//Dozowniki gotowe po jakiejkolwiek zmianie i któryś jest wybrany
VIS.bDispencersSyncReady :=	NOT tofDispencersSync.Q AND 
							(fbDispencer1Sync.bOut OR fbDispencer2Sync.bOut OR fbDispencer3Sync.bOut OR fbDispencer4Sync.bOut) AND
							(eDispencer1State = E_Station.eManualMovement OR NOT fbDispencer1Sync.bOut) AND
							(eDispencer2State = E_Station.eManualMovement OR NOT fbDispencer2Sync.bOut) AND
							(eDispencer3State = E_Station.eManualMovement OR NOT fbDispencer3Sync.bOut) AND
							(eDispencer4State = E_Station.eManualMovement OR NOT fbDispencer4Sync.bOut) 	
;
//Ustawianie dozowników
IF rtDispencer1Sync.Q THEN	bDispencer1DoSync	:= TRUE;END_IF
IF rtDispencer2Sync.Q THEN	bDispencer2DoSync	:= TRUE;END_IF
IF rtDispencer3Sync.Q THEN	bDispencer3DoSync	:= TRUE;END_IF
IF rtDispencer4Sync.Q THEN	bDispencer4DoSync	:= TRUE;END_IF

//Tylko w trybie serwisowym
IF bManualMode THEN
	
	IF VIS.bDispencersSyncReady THEN
	
		//Do wszystkich
		VIS.bDispencersHoming;	
		VIS.bDispencersManualDropCatcher;
		
		//Mycie
		VIS.bDispencer12Cleaning					:=	VIS.bDispencersCleaning						AND fbDispencer1Sync.bOut AND fbDispencer2Sync.bOut;
		VIS.bDispencer34Cleaning					:=	VIS.bDispencersCleaning						AND fbDispencer3Sync.bOut AND fbDispencer4Sync.bOut;

		//Podnośnik dozownika 1
		VIS.bDispencer12ManualLifterUp       		:=	VIS.bDispencersManualLifterUp       		AND (fbDispencer1Sync.bOut OR fbDispencer2Sync.bOut);		
		VIS.bDispencer12ManualLifterDown   			:=	VIS.bDispencersManualLifterDown   			AND (fbDispencer1Sync.bOut OR fbDispencer2Sync.bOut);	
		VIS.bDispencer12LifterStepMode				:=	VIS.bDispencersLifterStepMode				;	
		IF rtHeightSetDispencer12.Q THEN
			VIS.bDispencer12LifterHeightSet         :=	TRUE;
		END_IF		                                		

		//Dozownik 1	
		VIS.bDispencer1Dose                			:=	VIS.bDispencersDose                			AND fbDispencer1Sync.bOut;		
		VIS.bDispencer1IgnoreErrors        			:=	VIS.bDispencersIgnoreErrors        			AND fbDispencer1Sync.bOut;				
		VIS.bDispencer1ManualPistonBack     		:=	VIS.bDispencersManualPistonBack     		AND fbDispencer1Sync.bOut;		
		VIS.bDispencer1ManualPistonForward  		:=	VIS.bDispencersManualPistonForward  		AND fbDispencer1Sync.bOut;
		IF fbDispencer1Sync.bOut THEN					VIS.lrDispencersActPos 							:= VIS.lrDispencer1ActPos; 			END_IF
		IF fbDispencer1Sync.bOut THEN					VIS.lrDispencersLifterActPos      				:=	VIS.lrDispencer12LifterActPos ; END_IF	
		VIS.bDispencer1PullingFast          		:=	VIS.bDispencersPullingFast          		AND fbDispencer1Sync.bOut;		
		VIS.bDispencer1PullingSlow         			:=	VIS.bDispencersPullingSlow         			AND fbDispencer1Sync.bOut;		
		VIS.bDispencer1ManualSuckValve     			:=	VIS.bDispencersManualSuckValve     			AND fbDispencer1Sync.bOut;		
		VIS.bDispencer1ManualDoseValve     			:=	VIS.bDispencersManualDoseValve     			AND fbDispencer1Sync.bOut;
		VIS.lrDispencer12LifterSetPosStepMode		:=	VIS.lrDispencersLifterSetPosStepMode;	
		//Ready position					    	:=	//Ready position					    	AND fbDispencer1Sync.bOut;		

		//Dozownik 2 	
		VIS.bDispencer2Dose                			:=	VIS.bDispencersDose                			AND fbDispencer2Sync.bOut;		
		VIS.bDispencer2IgnoreErrors        			:=	VIS.bDispencersIgnoreErrors        			AND fbDispencer2Sync.bOut;				
		VIS.bDispencer2ManualPistonBack     		:=	VIS.bDispencersManualPistonBack     		AND fbDispencer2Sync.bOut;		
		VIS.bDispencer2ManualPistonForward  		:=	VIS.bDispencersManualPistonForward  		AND fbDispencer2Sync.bOut;
		IF fbDispencer2Sync.bOut THEN					VIS.lrDispencersActPos 							:= VIS.lrDispencer2ActPos; 			END_IF
		IF fbDispencer2Sync.bOut THEN					VIS.lrDispencersLifterActPos      				:=	VIS.lrDispencer12LifterActPos ; END_IF	
		VIS.bDispencer2PullingFast          		:=	VIS.bDispencersPullingFast          		AND fbDispencer2Sync.bOut;		
		VIS.bDispencer2PullingSlow         			:=	VIS.bDispencersPullingSlow         			AND fbDispencer2Sync.bOut;		
		VIS.bDispencer2ManualSuckValve     			:=	VIS.bDispencersManualSuckValve     			AND fbDispencer2Sync.bOut;		
		VIS.bDispencer2ManualDoseValve     			:=	VIS.bDispencersManualDoseValve     			AND fbDispencer2Sync.bOut;
		VIS.lrDispencer12LifterSetPosStepMode		:=	VIS.lrDispencersLifterSetPosStepMode;	                 
		//Ready position					    	:=	//Ready position					    	AND fbDispencer2Sync.bOut;		
		
		//Podnośnik dozownika 34
		VIS.bDispencer34ManualLifterUp       		:=	VIS.bDispencersManualLifterUp       		AND (fbDispencer3Sync.bOut OR fbDispencer4Sync.bOut);		
		VIS.bDispencer34ManualLifterDown   			:=	VIS.bDispencersManualLifterDown   			AND (fbDispencer3Sync.bOut OR fbDispencer4Sync.bOut);	
		VIS.bDispencer34LifterStepMode				:=	VIS.bDispencersLifterStepMode				;		
		IF rtHeightSetDispencer34.Q THEN
			VIS.bDispencer34LifterHeightSet         :=	TRUE;
		END_IF		
		//Dozownik 3 	
		VIS.bDispencer3Dose                			:=	VIS.bDispencersDose                			AND fbDispencer3Sync.bOut;		
		VIS.bDispencer3IgnoreErrors        			:=	VIS.bDispencersIgnoreErrors        			AND fbDispencer3Sync.bOut;				
		VIS.bDispencer3ManualPistonBack     		:=	VIS.bDispencersManualPistonBack     		AND fbDispencer3Sync.bOut;		
		VIS.bDispencer3ManualPistonForward  		:=	VIS.bDispencersManualPistonForward  		AND fbDispencer3Sync.bOut;
		IF fbDispencer3Sync.bOut THEN					VIS.lrDispencersActPos 							:= VIS.lrDispencer3ActPos; 			END_IF
		IF fbDispencer3Sync.bOut THEN					VIS.lrDispencersLifterActPos      				:=	VIS.lrDispencer34LifterActPos ; END_IF	
		VIS.bDispencer3PullingFast          		:=	VIS.bDispencersPullingFast          		AND fbDispencer3Sync.bOut;		
		VIS.bDispencer3PullingSlow         			:=	VIS.bDispencersPullingSlow         			AND fbDispencer3Sync.bOut;		
		VIS.bDispencer3ManualSuckValve     			:=	VIS.bDispencersManualSuckValve     			AND fbDispencer3Sync.bOut;		
		VIS.bDispencer3ManualDoseValve     			:=	VIS.bDispencersManualDoseValve     			AND fbDispencer3Sync.bOut;
		VIS.lrDispencer34LifterSetPosStepMode		:=	VIS.lrDispencersLifterSetPosStepMode;	                 
		//Ready position					    	:=	//Ready position					    	AND fbDispencer3Sync.bOut;		
	                           		
		//Dozownik 4 	
		VIS.bDispencer4Dose                			:=	VIS.bDispencersDose                			AND fbDispencer4Sync.bOut;		
		VIS.bDispencer4IgnoreErrors        			:=	VIS.bDispencersIgnoreErrors        			AND fbDispencer4Sync.bOut;				
		VIS.bDispencer4ManualPistonBack     		:=	VIS.bDispencersManualPistonBack     		AND fbDispencer4Sync.bOut;		
		VIS.bDispencer4ManualPistonForward  		:=	VIS.bDispencersManualPistonForward  		AND fbDispencer4Sync.bOut;
		IF fbDispencer4Sync.bOut THEN					VIS.lrDispencersActPos 							:= VIS.lrDispencer4ActPos; 			END_IF
		IF fbDispencer4Sync.bOut THEN					VIS.lrDispencersLifterActPos      				:=	VIS.lrDispencer34LifterActPos ; END_IF	
		VIS.bDispencer4PullingFast          		:=	VIS.bDispencersPullingFast          		AND fbDispencer4Sync.bOut;		
		VIS.bDispencer4PullingSlow         			:=	VIS.bDispencersPullingSlow         			AND fbDispencer4Sync.bOut;		
		VIS.bDispencer4ManualSuckValve     			:=	VIS.bDispencersManualSuckValve     			AND fbDispencer4Sync.bOut;		
		VIS.bDispencer4ManualDoseValve     			:=	VIS.bDispencersManualDoseValve     			AND fbDispencer4Sync.bOut;
		VIS.lrDispencer34LifterSetPosStepMode		:=	VIS.lrDispencersLifterSetPosStepMode;	                 
		//Ready position					    	:=	//Ready position					    	AND fbDispencer4Sync.bOut;		
			
	ELSE
		
		VIS.bDispencer1Dose                			:=	VIS.bDispencersDose    					 := FALSE;            			
		VIS.bDispencer1ManualPistonBack     		:=	VIS.bDispencersManualPistonBack     	 := FALSE;  
		VIS.bDispencer1ManualPistonForward  		:=	VIS.bDispencersManualPistonForward  	 := FALSE;  
		VIS.lrDispencersActPos 						:=	1234;			
		VIS.bDispencer12ManualLifterUp       		:=	VIS.bDispencersManualLifterUp       	 := FALSE;  	
		VIS.bDispencer12ManualLifterDown   			:=	VIS.bDispencersManualLifterDown   		 := FALSE;  
		VIS.lrDispencersLifterActPos      			:=	1234;		
		VIS.bDispencer1PullingFast          		:=	VIS.bDispencersPullingFast          	 := FALSE;  
		VIS.bDispencer1PullingSlow         			:=	VIS.bDispencersPullingSlow         		 := FALSE;  
		VIS.bDispencer1ManualSuckValve     			:=	VIS.bDispencersManualSuckValve     		 := FALSE;  
		VIS.bDispencer1ManualDoseValve     			:=	VIS.bDispencersManualDoseValve     		 := FALSE;  
		VIS.lrDispencer12LifterSetPosStepMode		:=	VIS.lrDispencersLifterSetPosStepMode	 := 2;	
		VIS.bDispencer12LifterStepMode				:=	VIS.bDispencersLifterStepMode		 	 := FALSE;  	
		//Ready position					    	:=	//Ready position					    
		//nie nadpisywać (bazownaie) VIS.bDispencer12LifterHeightSet          			:=	VIS.bDispencersHeightSet          		 := FALSE;  
		
		VIS.bDispencer2Dose                			:=	VIS.bDispencersDose    					 := FALSE;            			
		VIS.bDispencer2ManualPistonBack     		:=	VIS.bDispencersManualPistonBack     	 := FALSE;  
		VIS.bDispencer2ManualPistonForward  		:=	VIS.bDispencersManualPistonForward  	 := FALSE;  
		VIS.lrDispencersActPos 						:=	1234;			
		VIS.bDispencer12ManualLifterUp       		:=	VIS.bDispencersManualLifterUp       	 := FALSE;  	
		VIS.bDispencer12ManualLifterDown   			:=	VIS.bDispencersManualLifterDown   		 := FALSE;  
		VIS.lrDispencersLifterActPos      			:=	1234;		
		VIS.bDispencer2PullingFast          		:=	VIS.bDispencersPullingFast          	 := FALSE;  
		VIS.bDispencer2PullingSlow         			:=	VIS.bDispencersPullingSlow         		 := FALSE;  
		VIS.bDispencer2ManualSuckValve     			:=	VIS.bDispencersManualSuckValve     		 := FALSE;  
		VIS.bDispencer2ManualDoseValve     			:=	VIS.bDispencersManualDoseValve     		 := FALSE;  
		VIS.lrDispencer12LifterSetPosStepMode		:=	VIS.lrDispencersLifterSetPosStepMode	 := 2;	
		VIS.bDispencer12LifterStepMode				:=	VIS.bDispencersLifterStepMode		 	 := FALSE;  	
		//Ready position					    	:=	//Ready position					    
		 		
		VIS.bDispencer3Dose                			:=	VIS.bDispencersDose   					 := FALSE;            			
		VIS.bDispencer3ManualPistonBack     		:=	VIS.bDispencersManualPistonBack     	 := FALSE;  
		VIS.bDispencer3ManualPistonForward  		:=	VIS.bDispencersManualPistonForward  	 := FALSE;  
		VIS.lrDispencersActPos 						:=	1234;			
		VIS.bDispencer34ManualLifterUp       		:=	VIS.bDispencersManualLifterUp       	 := FALSE;  	
		VIS.bDispencer34ManualLifterDown   			:=	VIS.bDispencersManualLifterDown   		 := FALSE;  
		VIS.lrDispencersLifterActPos      			:=	1234;		
		VIS.bDispencer3PullingFast          		:=	VIS.bDispencersPullingFast          	 := FALSE;  
		VIS.bDispencer3PullingSlow         			:=	VIS.bDispencersPullingSlow         		 := FALSE;  
		VIS.bDispencer3ManualSuckValve     			:=	VIS.bDispencersManualSuckValve     		 := FALSE;  
		VIS.bDispencer3ManualDoseValve     			:=	VIS.bDispencersManualDoseValve     		 := FALSE;  
		VIS.lrDispencer34LifterSetPosStepMode		:=	VIS.lrDispencersLifterSetPosStepMode	 := 2;	
		VIS.bDispencer34LifterStepMode				:=	VIS.bDispencersLifterStepMode		 	 := FALSE;  	
		//Ready position					    	:=	//Ready position					    
		//VIS.bDispencer34LifterHeightSet          	:=	VIS.bDispencersHeightSet          		 := FALSE;  

		VIS.bDispencer4Dose                			:=	VIS.bDispencersDose    					 := FALSE;            			
		VIS.bDispencer4ManualPistonBack     		:=	VIS.bDispencersManualPistonBack     	 := FALSE;  
		VIS.bDispencer4ManualPistonForward  		:=	VIS.bDispencersManualPistonForward  	 := FALSE;  
		VIS.lrDispencersActPos 						:=	1234;			
		VIS.bDispencer34ManualLifterUp       		:=	VIS.bDispencersManualLifterUp       	 := FALSE;  	
		VIS.bDispencer34ManualLifterDown   			:=	VIS.bDispencersManualLifterDown   		 := FALSE;  
		VIS.lrDispencersLifterActPos      			:=	1234;		
		VIS.bDispencer4PullingFast          		:=	VIS.bDispencersPullingFast          	 := FALSE;  
		VIS.bDispencer4PullingSlow         			:=	VIS.bDispencersPullingSlow         		 := FALSE;  
		VIS.bDispencer4ManualSuckValve     			:=	VIS.bDispencersManualSuckValve     		 := FALSE;  
		VIS.bDispencer4ManualDoseValve     			:=	VIS.bDispencersManualDoseValve     		 := FALSE;  
		VIS.lrDispencer34LifterSetPosStepMode		:=	VIS.lrDispencersLifterSetPosStepMode	 := 2;	
		VIS.bDispencer34LifterStepMode				:=	VIS.bDispencersLifterStepMode		 	 := FALSE;  	
		//Ready position					    	:=	//Ready position					    
		
	END_IF
	
END_IF


(********KASOWANIE ROZKAZÓW CYKLI*********)
IF fbDispencer1.bCycleDone AND bManualMode AND
	(NOT fbDispencer2Sync.bOut AND NOT fbDispencer3Sync.bOut AND NOT fbDispencer4Sync.bOut)
THEN
    VIS.bDispencer1Dose := VIS.bDispencersDose :=  FALSE;
END_IF

IF fbDispencer2.bCycleDone AND bManualMode AND
	(NOT fbDispencer1Sync.bOut AND NOT fbDispencer3Sync.bOut AND NOT fbDispencer4Sync.bOut)
THEN
    VIS.bDispencer2Dose		:= VIS.bDispencersDose := FALSE;
END_IF

IF fbDispencer3.bCycleDone AND bManualMode AND
	(NOT fbDispencer1Sync.bOut AND NOT fbDispencer2Sync.bOut AND NOT fbDispencer4Sync.bOut)
THEN
    VIS.bDispencer3Dose		:= VIS.bDispencersDose := FALSE;
END_IF

IF fbDispencer4.bCycleDone AND bManualMode AND
	(NOT fbDispencer1Sync.bOut AND NOT fbDispencer2Sync.bOut AND NOT fbDispencer3Sync.bOut)

THEN
    VIS.bDispencer4Dose	:= VIS.bDispencersDose := FALSE;
END_IF
IF fbDispencer1.bCycleDone AND  fbDispencer2.bCycleDone AND NOT fbDispencer3.bCycleDone AND NOT fbDispencer4.bCycleDone AND bManualMode AND
	(fbDispencer1Sync.bOut AND fbDispencer2Sync.bOut AND NOT fbDispencer3Sync.bOut AND NOT fbDispencer4Sync.bOut)
THEN
    VIS.bDispencersDose :=  FALSE;
END_IF
IF NOT fbDispencer1.bCycleDone AND  NOT fbDispencer2.bCycleDone AND fbDispencer3.bCycleDone AND fbDispencer4.bCycleDone AND bManualMode AND
	(NOT fbDispencer1Sync.bOut AND NOT fbDispencer2Sync.bOut AND fbDispencer3Sync.bOut AND fbDispencer4Sync.bOut)
THEN
    VIS.bDispencersDose :=  FALSE;
END_IF
IF fbDispencer1.bCycleDone AND  fbDispencer2.bCycleDone AND  fbDispencer3.bCycleDone AND  fbDispencer4.bCycleDone AND bManualMode AND
	(fbDispencer1Sync.bOut AND fbDispencer2Sync.bOut AND fbDispencer3Sync.bOut AND fbDispencer4Sync.bOut)
THEN
    VIS.bDispencersDose :=  FALSE;
END_IF


(*****KONIEC KASOWANIA ROZKAZÓW CYKLI*****)
END_ACTION

ACTION aDosingChartHMI:
 fbDosingChart1(
	bWrite:= VIS.bDispencer1Dose, 
	nCycleTime:= 5, 
	lrData1:= VIS.lrDispencer1ActPos, 
	lrData2:= VIS.lrDispencer12LifterActPos, 
	bData3:= P02_Dispencers.QbDispencer1SuckingValveActuator, 
	bData4:= P02_Dispencers.QbDispencer1DosingValveActuator,
	bData5:= P02_Dispencers.QbDispencer1DropCatcherValveActuator,
	AsData=>VIS.AsChartDose1 );
	
 fbDosingStChart1(
	bWrite:= VIS.bDispencer1Dose, 
	udiCycleTime:= 5,
	lrAiData0:= VIS.lrDispencer1ActPos,
	lrAiData1:= VIS.lrDispencer12LifterActPos, 
	lrAiData2:= BOOL_TO_LREAL(P02_Dispencers.QbDispencer1SuckingValveActuator),
	lrAiData3:= BOOL_TO_LREAL(P02_Dispencers.QbDispencer1DosingValveActuator), 
	lrAiData4:= BOOL_TO_LREAL(P02_Dispencers.QbDispencer1DropCatcherValveActuator), 
	AiData=> VIS.AStAsChartDose1[0] );

fbDosingChart2(
	bWrite:= VIS.bDispencer2Dose, 
	nCycleTime:= 5, 
	lrData1:= VIS.lrDispencer2ActPos, 
	lrData2:= VIS.lrDispencer12LifterActPos, 
	bData3:= P02_Dispencers.QbDispencer2SuckingValveActuator, 
	bData4:= P02_Dispencers.QbDispencer2DosingValveActuator,
	bData5:= P02_Dispencers.QbDispencer2DropCatcherValveActuator,
	AsData=>VIS.AsChartDose2 );

 fbDosingStChart2(
	bWrite:= VIS.bDispencer1Dose, 
	udiCycleTime:= 5,
	lrAiData0:= VIS.lrDispencer2ActPos,
	lrAiData1:= VIS.lrDispencer12LifterActPos, 
	lrAiData2:= BOOL_TO_LREAL(P02_Dispencers.QbDispencer2SuckingValveActuator),
	lrAiData3:= BOOL_TO_LREAL(P02_Dispencers.QbDispencer2DosingValveActuator), 
	lrAiData4:= BOOL_TO_LREAL(P02_Dispencers.QbDispencer2DropCatcherValveActuator), 
	AiData=> VIS.AStAsChartDose2[0] );
	
fbDosingChart3(
	bWrite:= VIS.bDispencer3Dose, 
	nCycleTime:= 5,//nChartCycleTime, 
	lrData1:= VIS.lrDispencer3ActPos, 
	lrData2:= VIS.lrDispencer34LifterActPos, 
	bData3:= P02_Dispencers.QbDispencer3SuckingValveActuator, 
	bData4:= P02_Dispencers.QbDispencer3DosingValveActuator,
	bData5:= P02_Dispencers.QbDispencer3DropCatcherValveActuator,
	AsData=>VIS.AsChartDose3 );
	
 fbDosingStChart3(
	bWrite:= VIS.bDispencer1Dose, 
	udiCycleTime:= 5,
	lrAiData0:= VIS.lrDispencer3ActPos,
	lrAiData1:= VIS.lrDispencer34LifterActPos, 
	lrAiData2:= BOOL_TO_LREAL(P02_Dispencers.QbDispencer3SuckingValveActuator),
	lrAiData3:= BOOL_TO_LREAL(P02_Dispencers.QbDispencer3DosingValveActuator), 
	lrAiData4:= BOOL_TO_LREAL(P02_Dispencers.QbDispencer3DropCatcherValveActuator), 
	AiData=> VIS.AStAsChartDose3[0] );

fbDosingChart4(
	bWrite:= VIS.bDispencer4Dose, 
	nCycleTime:= 5,//nChartCycleTime, 
	lrData1:= VIS.lrDispencer4ActPos, 
	lrData2:= VIS.lrDispencer34LifterActPos, 
	bData3:= P02_Dispencers.QbDispencer4SuckingValveActuator, 
	bData4:= P02_Dispencers.QbDispencer4DosingValveActuator,
	bData5:= P02_Dispencers.QbDispencer4DropCatcherValveActuator,
	AsData=>VIS.AsChartDose4 );

fbDosingStChart4(
	bWrite:= VIS.bDispencer1Dose, 
	udiCycleTime:= 5,
	lrAiData0:= VIS.lrDispencer4ActPos,
	lrAiData1:= VIS.lrDispencer34LifterActPos, 
	lrAiData2:= BOOL_TO_LREAL(P02_Dispencers.QbDispencer4SuckingValveActuator),
	lrAiData3:= BOOL_TO_LREAL(P02_Dispencers.QbDispencer4DosingValveActuator), 
	lrAiData4:= BOOL_TO_LREAL(P02_Dispencers.QbDispencer4DropCatcherValveActuator), 
	AiData=> VIS.AStAsChartDose4[0] );
END_ACTION

ACTION aDropCatcher:
(**Uruchamianie ssawki tacek**)
P02_Dispencers.QbDispencerDropCatcherSuck;
IF (P00_PackML.fbPMLAuto.ePMLState = E_PMLState.ePMLState_EXECUTE OR P00_PackML.fbPMLModeManager.eModeStatus = E_PMLUnitMode.ePMLUnitMode_MANUAL) THEN
	fbDropCatcherSuck(T1:=T#5S , T0:=T#30S , Q=>P02_Dispencers.QbDispencerDropCatcherSuck);
	;
ELSE
	P02_Dispencers.QbDispencerDropCatcherSuck := FALSE;
END_IF

IF VIS.bDispencerManualDropCatcherSuck AND bManualMode THEN
	
	P02_Dispencers.QbDispencerDropCatcherSuck	:= TRUE;
END_IF
END_ACTION

ACTION aExSensor:


(** Czujnik Ex w zbiorniku **)

tonLowLevelExSensor(IN:=NOT IbTankLevelHighEX AND IbTankLevelLowEX AND NOT tonErrorExSensorDelay.Q AND bExEnable, PT:=T#1S);

IF tonLowLevelExSensor.Q THEN
	bTank1LevelExSensor:=TRUE;
ELSE
	bTank1LevelExSensor:=FALSE;
END_IF





//Błąd czujnika Ex
tonErrorExSensorDelay(IN:=IbTankLevelExError, PT:=T#5S);

IF tonErrorExSensorDelay.Q AND NOT TanksError.bError AND bExEnable AND bTank1SupplyPumpEnable THEN
	TanksError.bError:=TRUE;
	TanksError.bReset:=FALSE;
	TanksError.udiStationID:=78;
	TanksError.nErrorCode:=368;
	TanksError.sStationName:='Błąd systemu';
	TanksError.sErrorString:='Błąd czujnika poziomu Ex w zbiorniku. Sprawdz podłączenie lub stan separatora';
END_IF
END_ACTION

ACTION aLevelSensorCalibration:


(*
	bDialogBoxOn:BOOL;						(**)		// Wyświetlanie okienka komunikatów
	bDialogBoxText:STRING;					(**)		// Treść na oknie komunikatów
	bDialogBoxAck:BOOL;						(*t*)		// Potwierdzenie ogólne
	bDialogBoxCancelAck:BOOL;				(*t*)		// Wycofywanie procedury
	nDialogBoxType:UINT;								// Rodzaj okna, 0-nic, 1-tylko przysisk OK, 2 - tylko przycisk Anuluj, 3 - Przycisk OK i Anuluj
*)


(****Kalibracja czujnika nr 1 na pusto****)
tonTankLevelSensorCalibrationLight(IN:= nCalibrationDialog = 1 AND (VIS.bTank1LevelSensorCalibrationLight),PT:=T#10S);
tonTankLevelSensorCalibrationDark(IN:= nCalibrationDialog = 1 AND (VIS.bTank1LevelSensorCalibrationDark), PT:=T#5S);
IF VIS.bTank1LevelSensorCalibrationLight OR VIS.bTank1LevelSensorCalibrationDark THEN 		//Rozpoczaecie procedury kalibracji
	CASE nCalibrationDialog OF
		
		0: //Pytanie Czy na pewno
			VIS.nDialogBoxType	:=	3;									//Wyświetlanie przycisku OK i Anuluj
			IF VIS.bTank1LevelSensorCalibrationLight THEN
				VIS.bDialogBoxText	:=	'Want calibrate the level sensor to an empty tank? Immerse the sensor in the mass and remove it, simulating an empty tank.';
				VIS.sDialogBoxPicture	:= 'info';
			ELSIF VIS.bTank1LevelSensorCalibrationDark THEN
				VIS.bDialogBoxText	:=	'Should I calibrate the level sensor to a full tank? Immerse the sensor in the mass to simulate a full tank.';
				VIS.sDialogBoxPicture	:= 'info';
			END_IF
			VIS.bDialogBoxOn	:=	TRUE;
			IF VIS.bDialogBoxAck THEN
				VIS.bDialogBoxAck	:=	FALSE;		
				nCalibrationDialog:=nCalibrationDialog+1;
			ELSIF VIS.bDialogBoxCancelAck THEN
				VIS.bTank1LevelSensorCalibrationLight	:=	FALSE;
				VIS.bTank1LevelSensorCalibrationDark	:=	FALSE;

				//MAIN.aResetDialog();	
				nCalibrationDialog := 0;
			END_IF
			
		1: //Trwa kalibracja
			VIS.nDialogBoxType	:=	0;									//Bez przycisków
			
			IF VIS.bTank1LevelSensorCalibrationLight THEN
				QbTank1LevelSensorCalibration := NOT tonTankLevelSensorCalibrationLight.Q;	
				VIS.bDialogBoxText	:=	'Empty tank calibration in progress 1...';
				VIS.sDialogBoxPicture	:= '';
			END_IF
			IF VIS.bTank1LevelSensorCalibrationDark THEN
				QbTank1LevelSensorCalibration := NOT tonTankLevelSensorCalibrationDark.Q;	
				VIS.bDialogBoxText	:=	'Full tank calibration in progress 1...';
				VIS.sDialogBoxPicture	:= '';
			END_IF
			IF tonTankLevelSensorCalibrationLight.Q OR tonTankLevelSensorCalibrationDark.Q THEN
				nCalibrationDialog:=nCalibrationDialog+1;
			END_IF
			
		2: //Koniec kalibracji
			VIS.nDialogBoxType	:=	1;									//Potwierdz kalibracje
			VIS.bDialogBoxText	:=	'Calibration completed successfully';
			VIS.sDialogBoxPicture	:= 'ok';
			IF VIS.bTank1LevelSensorCalibrationLight OR VIS.bTank1LevelSensorCalibrationDark THEN
				bTank1LevelSensorCalibrated := TRUE;						//Zmienna presistent o kalibracji
			END_IF
			
			IF  VIS.bDialogBoxAck THEN
				VIS.bDialogBoxAck :=					FALSE;
				VIS.bTank1LevelSensorCalibrationLight	:=	FALSE;
				VIS.bTank1LevelSensorCalibrationDark	:=	FALSE;
				P00_Visualization.aResetDialog();
				nCalibrationDialog := 0;
			END_IF
			
	END_CASE
END_IF
END_ACTION

ACTION aLimits:

(*Zabezpieczenie nastaw dozowników*)
//Dozownika 1 i 2 (1 faza)
IF VIS.lrDispencer1DoseValveOpenTimeAccShow>0 			THEN 	VIS.lrDispencer1DoseValveOpenVolumeShow		:=0;		END_IF
IF VIS.lrDispencer1DoseValveCloseTimeDecShow>0 			THEN	VIS.lrDispencer1DoseValveCloseVolumeShow	:=0;		END_IF
IF VIS.bDispencer1DoseSuckingShow 						THEN	VIS.lrDispencer1DoseValveCloseVolumeShow	:=0;		END_IF
IF VIS.lrDispencer1SuckValveOpenTimeDelayShow>0 		THEN	VIS.lrDispencer1SuckValveOpenVolumeShow		:=0;		END_IF
IF VIS.lrDispencer1SuckValveCloseTimeDelayShow>0 		THEN	VIS.lrDispencer1SuckValveCloseVolumeShow	:=0;		END_IF
IF VIS.lrDispencer1Phase1VolumeShow > VIS.lrDispencer1DoseVolumeShow - VIS.lrDispencer1Phase2VolumeShow THEN	VIS.lrDispencer1Phase1VolumeShow	:= VIS.lrDispencer1DoseVolumeShow - VIS.lrDispencer1Phase2VolumeShow;END_IF
IF VIS.lrDispencer1Phase2VolumeShow > VIS.lrDispencer1DoseVolumeShow - VIS.lrDispencer1Phase1VolumeShow THEN	VIS.lrDispencer1Phase2VolumeShow 	:= VIS.lrDispencer1DoseVolumeShow - VIS.lrDispencer1Phase1VolumeShow;END_IF
IF VIS.lrDispencer1Phase2VolumeShow > VIS.lrDispencer1DoseVolumeShow 									THEN	VIS.lrDispencer1Phase1VolumeShow	:= 0;	VIS.lrDispencer1Phase2VolumeShow 	:= VIS.lrDispencer1DoseVolumeShow;END_IF

// Dozownika 3 i 4 (2 faza)
IF VIS.lrDispencer2DoseValveOpenTimeAccShow>0 			THEN	VIS.lrDispencer2DoseValveOpenVolumeShow		:=0;		END_IF
IF VIS.lrDispencer2DoseValveCloseTimeDecShow>0 			THEN	VIS.lrDispencer2DoseValveCloseVolumeShow	:=0;		END_IF
IF VIS.bDispencer2DoseSuckingShow 						THEN	VIS.lrDispencer2DoseValveCloseVolumeShow	:=0;		END_IF
IF VIS.lrDispencer2SuckValveOpenTimeDelayShow>0 		THEN	VIS.lrDispencer2SuckValveOpenVolumeShow		:=0;		END_IF
IF VIS.lrDispencer2SuckValveCloseTimeDelayShow>0 		THEN	VIS.lrDispencer2SuckValveCloseVolumeShow	:=0;		END_IF
IF VIS.lrDispencer2Phase1VolumeShow > VIS.lrDispencer2DoseVolumeShow - VIS.lrDispencer2Phase2VolumeShow THEN	VIS.lrDispencer2Phase1VolumeShow	:= VIS.lrDispencer2DoseVolumeShow - VIS.lrDispencer2Phase2VolumeShow;END_IF
IF VIS.lrDispencer2Phase2VolumeShow > VIS.lrDispencer2DoseVolumeShow - VIS.lrDispencer2Phase1VolumeShow THEN	VIS.lrDispencer2Phase2VolumeShow 	:= VIS.lrDispencer2DoseVolumeShow - VIS.lrDispencer2Phase1VolumeShow;END_IF
IF VIS.lrDispencer2Phase2VolumeShow > VIS.lrDispencer2DoseVolumeShow 									THEN	VIS.lrDispencer2Phase1VolumeShow	:= 0;	VIS.lrDispencer2Phase2VolumeShow 	:= VIS.lrDispencer2DoseVolumeShow;END_IF

IF lrDispencersLifterReadyPosition <1 					THEN	lrDispencersLifterReadyPosition			:=	270;													END_IF
IF 	VIS.lrDispencersLifterReadyPositionShow > 
	(P02_Dispencers.fbDispencer1.lrMaxPosition - 2)		THEN	VIS.lrDispencersLifterReadyPositionShow	:=	P02_Dispencers.fbDispencer1.lrMaxPosition - 2;			END_IF
	
	
IF 	VIS.lrFormsDragingLeftStartPosition		= 0		THEN	VIS.lrFormsDragingLeftStartPosition		:=	7;		END_IF;
IF 	VIS.lrFormsDragingLeftEndPosition		= 0		THEN	VIS.lrFormsDragingLeftEndPosition		:=	137;	END_IF;
IF 	VIS.lrFormsDragingRightStartPosition	= 0		THEN	VIS.lrFormsDragingRightStartPosition	:=	7.5;		END_IF;
IF 	VIS.lrFormsDragingRightEndPosition		= 0		THEN	VIS.lrFormsDragingRightEndPosition		:=	139;	END_IF;;
END_ACTION

ACTION aTankHeating:
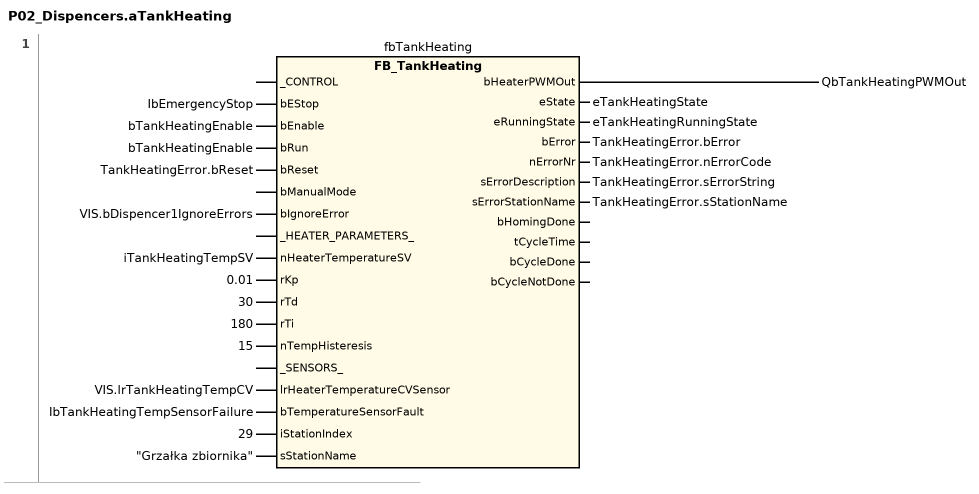
// NETWORK 1
fbTankHeating(
    bEStop := IbEmergencyStop,
    bEnable := bTankHeatingEnable,
    bRun := bTankHeatingEnable,
    bReset := TankHeatingError.bReset,
    bIgnoreError := VIS.bDispencer1IgnoreErrors,
    nHeaterTemperatureSV := iTankHeatingTempSV,
    rKp := 0.01,
    rTd := 30,
    rTi := 180,
    nTempHisteresis := 15,
    lrHeaterTemperatureCVSensor := VIS.lrTankHeatingTempCV,
    bTemperatureSensorFault := IbTankHeatingTempSensorFailure,
    iStationIndex := 29,
    sStationName := "Grzałka zbiornika",
    eState => eTankHeatingState,
    eRunningState => eTankHeatingRunningState,
    bError => TankHeatingError.bError,
    nErrorNr => TankHeatingError.nErrorCode,
    sErrorDescription => TankHeatingError.sErrorString,
    sErrorStationName => TankHeatingError.sStationName); // FB_TankHeating
QbTankHeatingPWMOut := fbTankHeating.bHeaterPWMOut;
END_ACTION

ACTION aTanks:
//Sterowanie Mieszadłem zbiornikowym
IF IbEmergencyStop (*AND IbFuseTankMixerEngineOK*) THEN
	QbTank1MixerStart:=(bTank1MixerEnable AND NOT bChangeover) OR (VIS.bTank1ManualMixer AND bManualMode);
ELSE
	QbTank1MixerStart:=FALSE;
	VIS.bTank1ManualMixer:=FALSE;
END_IF

//Sterowanie grzaniem zbiornika
//QbTank1HeaterOn:=IbEmergencyStopButton AND bTank1HeaterEnable OR (VIS.bManualTank1Heater AND bManualMode);

//Odwracanie sygnałów z czujników poziomu z receptur
bTank1LevelSignalInvert;									// Odwróć sygnał z czujnika zbiornika pierwszego
bTank2LevelSignalInvert;									// Odwróć sygnał z czujnika zbionirka drugiego
VIS.bTank1SupplyPumpEnableShow;
VIS.bTank2SupplyPumpEnableShow;
//Zmienne do poglądu zadziałania pomp od czujników
VIS.bHMITank1LevelSensorPumpOn;								// Sygnał z czujnika poziomu 1 załączający pompe 1 zależnie od ustawień (do podglądu sprawdzenia działania pompy bez jej załaczania)
VIS.bHMITank2LevelSensorPumpOn;								// Sygnał z czujnika poziomu 2 załączający pompe 2 zaleznie od ustawień (do podglądu sprawdzenia działania pompy bez jej załaczania)

//Odwracanie sygnałów z czujników poziomu
IF NOT bTank1LevelSignalInvert THEN
	bTank1LevelLow					:=	IbTank1LevelLow OR bTank1LevelLowConductiveSensor OR bTank1LevelExSensor; 	
	VIS.bHMITank1LevelSensorPumpOn	:=	IbTank1LevelLow OR bTank1LevelLowConductiveSensor OR bTank1LevelExSensor; 	
ELSE
	bTank1LevelLow					:=	NOT IbTank1LevelLow;
	VIS.bHMITank1LevelSensorPumpOn	:=	NOT IbTank1LevelLow;
END_IF
IF NOT bTank2LevelSignalInvert THEN
	bTank2LevelLow					:=	IbTank2LevelLow OR bTank2LevelLowConductiveSensor;
	VIS.bHMITank2LevelSensorPumpOn	:=	IbTank2LevelLow OR bTank2LevelLowConductiveSensor;
ELSE
	bTank2LevelLow					:=	NOT IbTank2LevelLow;	
	VIS.bHMITank2LevelSensorPumpOn	:=	NOT IbTank2LevelLow;
END_IF

// Mycie CIP

IF bCIP THEN
	tonTank1LevelSensor(IN:= bTank1LevelLow,PT:=T#15S);
ELSE
	IF VIS.lrDispencer1DoseVolumeShow > 450 THEN
		tonTank1LevelSensor(IN:= bTank1LevelLow,PT:=T#500MS);
	ELSE
		tonTank1LevelSensor(IN:= bTank1LevelLow,PT:=T#5S);		
	END_IF
END_IF
	
//Sterowanie pompą podającą nr 1
tofTank1LevelSensor(IN:= bTank1LevelLow,PT:=T#0S);

IF IbEmergencyStop AND (tofTank1LevelSensor.Q OR  tonTank1LevelSensor.Q) AND NOT GVL.SensorAcetoneError.bError AND NOT bHomingDialog THEN  // dodany sygnał od czujnika acetonu
	QbTank1PumpStart:=(bTank1SupplyPumpEnable AND NOT bChangeover) OR (VIS.bTank1ManualSupplyPump AND bManualMode);
ELSE
	QbTank1PumpStart:=FALSE;
END_IF

//Sterowanie pompą podającą nr 2
tofTank2LevelSensor(IN:= bTank2LevelLow,PT:=T#0S);
tonTank2LevelSensor(IN:= bTank2LevelLow,PT:=T#5S);
IF IbEmergencyStop AND (tofTank2LevelSensor.Q OR tonTank2LevelSensor.Q) AND NOT bHomingDialog THEN  // dodany sygnał od czujnika acetonu THEN
	QbTank2PumpStart:=(bTank2SupplyPumpEnable AND NOT bChangeover) OR (VIS.bTank2ManualSupplyPump AND bManualMode);
ELSE
	QbTank2PumpStart:=FALSE;
END_IF

//ERROR HANDLING
// Alarm_0100	100	Error	Zbiornik 1 | Brak masy w leju
// Alarm_0101	101	Error	Zbiornik 2 | Brak masy w leju
// Alarm_0102	102	Error	Mixer | Wyłączone zabezpieczenie przy próbie uruchomienia
// Alarm_0103	103	Error	Pompa 1 | Przepalony bezpiecznik - sprawdź połączenie i wymień
// Alarm_0104	104	Error	Pompa 2 | Przepalony bezpiecznik - sprawdź połączenie i wymień

IF bAlarmInit THEN
    bAlarmInit := FALSE; 
	fbSourceInfo.Clear();
	fbSourceInfo.sName:='Błąd systemu';//sStationName;//'Machine';
	fbSourceInfo.nId:=78;//udiStationID;//2700;
	// Alarm_0100	100	Error	Zbiornik 1 | Brak masy w leju
    arfbAlarm[0].CreateEx(stEventEntry := TC_EVENTS.AlarmClass.Alarm_0100, bWithConfirmation:= FALSE,  ipSourceInfo:= fbSourceInfo); 
	// Alarm_0101	101	Error	Zbiornik 2 | Brak masy w leju
	arfbAlarm[1].CreateEx(stEventEntry := TC_EVENTS.AlarmClass.Alarm_0101, bWithConfirmation:= FALSE,  ipSourceInfo:= fbSourceInfo); 
	// Alarm_0102	102	Error	Mixer | Wyłączone zabezpieczenie przy próbie uruchomienia
	arfbAlarm[2].CreateEx(stEventEntry := TC_EVENTS.AlarmClass.Alarm_0102, bWithConfirmation:= FALSE,  ipSourceInfo:= fbSourceInfo); 
	// Alarm_0103	103	Error	Pompa 1 | Przepalony bezpiecznik - sprawdź połączenie i wymień
	arfbAlarm[3].CreateEx(stEventEntry := TC_EVENTS.AlarmClass.Alarm_0103, bWithConfirmation:= FALSE,  ipSourceInfo:= fbSourceInfo); 
	// Alarm_0104	104	Error	Pompa 2 | Przepalony bezpiecznik - sprawdź połączenie i wymień
	arfbAlarm[4].CreateEx(stEventEntry := TC_EVENTS.AlarmClass.Alarm_0104, bWithConfirmation:= FALSE,  ipSourceInfo:= fbSourceInfo); 
END_IF


// Alarm_0100	100	Error	Zbiornik 1 | Brak masy w leju
//BŁĄD 72- Brak masy w leju	zbiorniku 1
//tonTank1EmptyAlarm(IN:=bTank1LevelLow AND (eMachineState=E_MachineState.eCycleOn OR eMachineState=E_MachineState.eCycleStarting OR eMachineState = E_MachineState.eConfectionEnd),PT:=T#25S);
//Opcja z liczeniem ilości doz
IF bTank1SupplyPumpEnable AND (tonTank1EmptyAlarm.Q OR nDose1CounterWhenLowLevel>=nDoseCounter1) AND NOT VIS.bTanksIgnoreError THEN
	IF NOT arfbAlarm[0].bActive THEN
			arfbAlarm[0].Raise(nTimeStamp:=0);
		END_IF
	ELSE	
		IF  arfbAlarm[0].bActive AND TanksError.bReset THEN
			arfbAlarm[0].Clear(nTimeStamp:=0, bResetConfirmation:= FALSE);
	END_IF	
// 	TanksError.bError:=TRUE;
// 	TanksError.bReset:=FALSE;
// 	TanksError.udiStationID:=78;
// 	TanksError.nErrorCode:=72;
// 	TanksError.sStationName:='Błąd systemu';
// 	TanksError.sErrorString:='Zbiornik 1 | Brak masy w leju';
END_IF
// Alarm_0101	101	Error	Zbiornik 2 | Brak masy w leju
//BŁĄD 73- Brak masy w leju	zbiorniku 2																	
//tonTank2EmptyAlarm(IN:=bTank2LevelLow AND (eMachineState=E_MachineState.eCycleOn OR eMachineState=E_MachineState.eCycleStarting OR eMachineState = E_MachineState.eConfectionEnd),PT:=T#25S);
//Opcja z liczeniem ilości doz
//tonTank2EmptyAlarm(IN:=(bTank2LevelLow OR nDose2CounterWhenLowLevel>=nDoseCounter2)	AND (P00_PackML.fbPMLAuto.ePMLState = E_PMLState.ePMLState_EXECUTE OR P00_PackML.fbPMLAuto.ePMLState = E_PMLState.ePMLState_STARTING),PT:=T#25S);
IF bTank2SupplyPumpEnable AND (tonTank2EmptyAlarm.Q OR nDose2CounterWhenLowLevel>=nDoseCounter1) AND NOT VIS.bTanksIgnoreError THEN
		IF NOT arfbAlarm[1].bActive THEN
			arfbAlarm[1].Raise(nTimeStamp:=0);
		END_IF
	ELSE	
		IF  arfbAlarm[1].bActive AND TanksError.bReset THEN
			arfbAlarm[1].Clear(nTimeStamp:=0, bResetConfirmation:= FALSE);
	END_IF
// 	TanksError.bError:=TRUE;
// 	TanksError.bReset:=FALSE;
// 	TanksError.udiStationID:=78;
// 	TanksError.nErrorCode:=73;
// 	TanksError.sStationName:='Błąd systemu';
// 	TanksError.sErrorString:='Zbiornik 2 | Brak masy w leju';
END_IF
// Alarm_0102	102	Error	Mixer | Wyłączone zabezpieczenie przy próbie uruchomienia
//BŁĄD 74- Błąd zabezpieczenia mieszadła podczas właczenia zasilania jednego
tonMixerNotWorking(IN:=NOT IbFuseTankMixerEngineOK AND QbTank1MixerStart, PT:=T#3S);
IF tonMixerNotWorking.Q THEN
		IF NOT arfbAlarm[2].bActive THEN
			arfbAlarm[2].Raise(nTimeStamp:=0);
		END_IF
	ELSE	
		IF  arfbAlarm[2].bActive AND TanksError.bReset THEN
			arfbAlarm[2].Clear(nTimeStamp:=0, bResetConfirmation:= FALSE);
	END_IF
// 	TanksError.bError:=TRUE;
// 	TanksError.bReset:=FALSE;
// 	TanksError.udiStationID:=78;
// 	TanksError.nErrorCode:=74;
// 	TanksError.sStationName:='Błąd systemu';
// 	TanksError.sErrorString:='Mixer | Wyłączone zabezpieczenie przy próbie uruchomienia';
END_IF
// Alarm_0103	103	Error	Pompa 1 | Przepalony bezpiecznik - sprawdź połączenie i wymień
//BŁĄD 75 - Przepalony bezpiecznik pompy 1 
tonTank1PumpFuseOK(IN:= QbTank1PumpStart AND NOT IbTank1PumpFuseOK, PT:= T#1S);
IF tonTank1PumpFuseOK.Q  THEN
		IF NOT arfbAlarm[3].bActive THEN
			arfbAlarm[3].Raise(nTimeStamp:=0);
		END_IF
	ELSE	
		IF  arfbAlarm[3].bActive AND TanksError.bReset THEN
			arfbAlarm[3].Clear(nTimeStamp:=0, bResetConfirmation:= FALSE);
	END_IF
// 	TanksError.bError:=TRUE;
// 	TanksError.bReset:=FALSE;
// 	TanksError.udiStationID:=78;
// 	TanksError.nErrorCode:=75;
// 	TanksError.sStationName:='Błąd systemu';
// 	TanksError.sErrorString:='Pompa 1 | Przepalony bezpiecznik - sprawdź połączenie i wymień';
END_IF
// Alarm_0104	104	Error	Pompa 2 | Przepalony bezpiecznik - sprawdź połączenie i wymień
//BŁĄD 76- Przepalony bezpiecznik pompy 2 
tonTank2PumpFuseOK(IN:= QbTank2PumpStart AND NOT IbTank2PumpFuseOK, PT:= T#1S);
IF tonTank2PumpFuseOK.Q THEN
		IF NOT arfbAlarm[4].bActive THEN
			arfbAlarm[4].Raise(nTimeStamp:=0);
		END_IF
	ELSE	
		IF  arfbAlarm[4].bActive AND TanksError.bReset THEN
			arfbAlarm[4].Clear(nTimeStamp:=0, bResetConfirmation:= FALSE);
	END_IF
// 	TanksError.bError:=TRUE;
// 	TanksError.bReset:=FALSE;
// 	TanksError.udiStationID:=78;
// 	TanksError.nErrorCode:=76;
// 	TanksError.sStationName:='Błąd systemu';
// 	TanksError.sErrorString:='Pompa 2 | Przepalony bezpiecznik - sprawdź połączenie i wymień';
END_IF



//BŁĄD 21- zaklejenie czujnika w zbiorniku	
rtDispencer1DoseDone(CLK:=P02_Dispencers.fbDispencer1.bCycleDone,Q=>);
rtDispencer2DoseDone(CLK:=P02_Dispencers.fbDispencer2.bCycleDone,Q=>);

IF bTank1LevelLow THEN
	nDose1Counter:=0;
ELSIF rtDispencer1DoseDone.Q THEN
	nDose1Counter:=nDose1Counter+1;
END_IF

IF bTank2LevelLow THEN
	nDose2Counter:=0;
ELSIF rtDispencer2DoseDone.Q THEN
	nDose2Counter:=nDose2Counter+1;
END_IF

IF rtDispencer1DoseDone.Q  AND bTank1LevelLow THEN
	nDose1CounterWhenLowLevel := nDose1CounterWhenLowLevel	+	1;
END_IF
IF rtDispencer2DoseDone.Q AND bTank2LevelLow THEN
	nDose2CounterWhenLowLevel := nDose2CounterWhenLowLevel	+	1;
END_IF
IF NOT bTank1LevelLow THEN
	nDose1CounterWhenLowLevel := 0;
END_IF
IF NOT bTank2LevelLow THEN
	nDose2CounterWhenLowLevel := 0;
END_IF

(*Obliczanie wartości liczby dozy po których jest alarm zależnie od dozy*)

IF NOT bDosingTwoPhases THEN
	IF lrDispencer1DoseVolume > 0 AND lrDispencer1DoseVolume < 300 THEN //Zawsze błąd po 2 litrach na jeden dozownik czyli 4 litry
		nDoseCounter1 := LREAL_TO_INT( 827 * EXPT(lrDispencer1DoseVolume,-0.959));
		//nDoseCounter1 := LREAL_TO_INT( 2467.3 * EXPT(lrDispencer1DoseVolume,-1.082));		
	ELSIF 	lrDispencer1DoseVolume > 600 THEN
		nDoseCounter1 := 4;
	ELSIF 	lrDispencer1DoseVolume > 450 THEN
		nDoseCounter1 := 8;
	ELSIF 	lrDispencer1DoseVolume > 300 THEN
		nDoseCounter1 := 13;		
	ELSE
		nDoseCounter1 := 25 ;
	END_IF
ELSE
	IF lrDispencer1DoseVolume > 0 THEN //Zawsze błąd po 2 litrach na jeden dozownik czyli 4 litry
		nDoseCounter1 := LREAL_TO_INT( 827 * EXPT(lrDispencer1DoseVolume,-0.959));
		//nDoseCounter1 := LREAL_TO_INT( 2467.3 * EXPT(lrDispencer1DoseVolume,-1.082));		
	ELSE
		nDoseCounter1 := 25 ;
	END_IF
	IF lrDispencer2DoseVolume > 0 THEN //Zawsze błąd po 2 litrach na jeden dozownik czyli 4 litry
		nDoseCounter2 := LREAL_TO_INT( 827 * EXPT(lrDispencer2DoseVolume,-0.959));
		//nDoseCounter2 := LREAL_TO_INT( 2467.3 * EXPT(lrDispencer2DoseVolume,-1.082));		
	ELSE
		nDoseCounter2 := 25 ;
	END_IF
END_IF
IF nDoseCounter1 < 3 THEN	nDoseCounter1 := 3;END_IF
IF nDoseCounter2 < 3 THEN	nDoseCounter2 := 3;END_IF

(*IF bTank1SupplyPumpEnable AND nDose1Counter>nDoseCounter1 AND NOT TanksError.bError AND NOT VIS.bTanksIgnoreError THEN
	TanksError.bError:=TRUE;
	TanksError.bReset:=FALSE;
	TanksError.nErrorCode:=22;
	TanksError.sStationName:='Zbiornik 1';
	TanksError.sErrorString:='Zaklejony czujnik w zbiorniku';
END_IF*)

(*IF bTank2SupplyPumpEnable AND nDose2Counter>nDoseCounter2 AND NOT TanksError.bError AND NOT VIS.bTanksIgnoreError THEN
	TanksError.bError:=TRUE;
	TanksError.bReset:=FALSE;
	TanksError.nErrorCode:=23;
	TanksError.sStationName:='Zbiornik 2';
	TanksError.sErrorString:='Zaklejony czujnik w zbiorniku';
END_IF*)

IF TanksError.bReset THEN
	nDose1CounterWhenLowLevel := 0;
	nDose2CounterWhenLowLevel := 0;
	nDose1Counter := 0;
	nDose2Counter := 0;
//	TanksError.bError:=FALSE;
//	TanksError.bReset:=FALSE;
//	TanksError.nErrorCode:=0;
//	TanksError.sStationName:='';
//	TanksError.sErrorString:='';
END_IF

(*Wyświetlanie błedu na wyjściu*)
TanksError.bError							:= FALSE;
FOR nAlarmNumerator := 0 TO 19 DO
	TanksError.bError						:= TanksError.bError OR arfbAlarm[nAlarmNumerator].bActive;
END_FOR

(***Ciśnienie w zbiornikach****)
P02_Dispencers.QbTank1Pressure:=(bTank1PressureEnable AND NOT bChangeover) OR (VIS.bTank1ManualPressure AND bManualMode);

(***WYŁĄCZANIE JEZELI NIE SA W TRYBIE SERWISOWYM***)
IF NOT bManualMode THEN
	VIS.bTank1ManualSupplyPump := FALSE;
	VIS.bTank2ManualSupplyPump := FALSE;
	VIS.bTank1ManualPressure := FALSE;
	VIS.bTank1ManualMixer := FALSE;
END_IF
END_ACTION

ACTION aTanksRainbowMode:
VIS.bTankRainbowModeShow;
bTankRainbowMode;

VIS.bHMITank3LevelSensorPumpOn;	
VIS.iTank3LevelSensorValue;		
VIS.bHMITank4LevelSensorPumpOn;	
VIS.iTank4LevelSensorValue;		

VIS.uTank1LevelSetpointShow;
VIS.uTank1LevelSetpointShow;
END_ACTION

ACTION aTankWarning:

(****Ostrzezenia***)
//Niski poziom w zbiorniku 1
tonTank1LevelWarning (IN:=	VIS.iTank1LevelSensorValue < 10 AND 
							P00_PackML.fbPMLAuto.ePMLState =	Tc3_PackML.E_PMLState.ePMLState_EXECUTE
					, PT:=T#3S);

IF tonTank1LevelWarning.Q AND NOT TanksWarning[0].bWarning THEN
	TanksWarning[0].bWarning									:=TRUE;
	TanksWarning[0].udiWarningCode								:=25;
	TanksWarning[0].sDescription								:= 'Zbiornik 1 | Niski poziom w zbiorniku';
ELSIF NOT tonTank1LevelWarning.Q AND TanksWarning[0].bAcknowledge THEN
	TanksWarning[0].bWarning									:=FALSE;
	TanksWarning[0].bAcknowledge								:=FALSE;
	VIS.uliWarningAcknowledge.0 								:=FALSE;
ELSIF TanksWarning[0].bAcknowledge THEN
	TanksWarning[0].bAcknowledge								:=TRUE;
END_IF

//Niski poziom w zbiorniku 2
tonTank1LevelWarning (IN:=	VIS.iTank2LevelSensorValue < 10 AND bDosingTwoPhases AND 
							P00_PackML.fbPMLAuto.ePMLState =	Tc3_PackML.E_PMLState.ePMLState_EXECUTE
					, PT:=T#3S);

IF tonTank1LevelWarning.Q AND NOT TanksWarning[1].bWarning THEN
	TanksWarning[1].bWarning									:=TRUE;
	TanksWarning[1].udiWarningCode								:=26;
	TanksWarning[1].sDescription								:= 'Zbiornik 2 | Niski poziom w zbiorniku';
ELSIF NOT tonTank1LevelWarning.Q AND TanksWarning[1].bAcknowledge THEN
	TanksWarning[1].bWarning									:=FALSE;
	TanksWarning[1].bAcknowledge								:=FALSE;
	VIS.uliWarningAcknowledge.1 								:=FALSE;
ELSIF TanksWarning[1].bAcknowledge THEN
	TanksWarning[1].bAcknowledge								:=TRUE;
END_IF
END_ACTION

ACTION aTDRMassSensor:
(*
Nazwa:			aTDRMassSensor
Opis:			Czujnik poziomu z prętem SICK 
Wersja:			v1.0
Data:			2021-05-17
Autor:			DP,MP
Urzadzenia:		Sick LFP
Konfiguracja:	
Info:
- przypisać zmienna od diagnostyki do blędów IO-LINK, żeby po wypięciu czujnika nie zaczeła pompowac pompa
- Ustawienia czujnika:
Parameter menu>PARAMETERS	>DspVAL-Distan
							>FIlter 400ms
				>EXPERT		>Mode Pulse
							>MeasMd HiAcc
							>MaxCol	10cm/s
				>Pulse		>TrsHld	50 NAJWAZNIEJSZE
							>CalRng 6005	
							>MaskZn 0
							>MaskTr 50
				>Probe		>Lenght 305
							>CblLen 1000
							>Type Rod
Kalibracja na pustym zbiorniku
SigQua musi byc powyżej 40 jeżeli wykrywa mase
Jeżeli nie wykrywa masy lub coś jest nie tak nalezy zwiększyć TrsHld
Za każdą zmianą trzeba kalibrowac czujnik
- Pompowanie zawsze do 150mm czujnika

*)


(*Przypisane na stałe*)
(*IF VIS.bTank1LevelSensorLow THEN // Poziom zależnie od nastaw
	VIS.uTank1LevelSetpointShow:=1;
ELSIF VIS.bTank1LevelSensorHigh THEN // Poziom zależnie od nastaw
	VIS.uTank1LevelSetpointShow:=120; //bylo 150
ELSE
	VIS.uTank1LevelSetpointShow:=140; //bylo 120
END_IF*)

IF VIS.uTank1LevelSetpointShow > 201 THEN
	VIS.uTank1LevelSetpointShow := 100;
END_IF



(**************************** ZBIORNIK 1***********************************************************)
(*Przypisanie zmiennych wizualiazji do zmiennych wewnetrznych programu*)
                     
iTank1Sensor1ValueTemp.0		:= 			IusiTank1SensorValue0.7		;
iTank1Sensor1ValueTemp.1		:= 			IusiTank1SensorValue0.6		;
iTank1Sensor1ValueTemp.2		:= 			IusiTank1SensorValue0.5		;
iTank1Sensor1ValueTemp.3		:= 			IusiTank1SensorValue0.4		;
iTank1Sensor1ValueTemp.4		:= 			IusiTank1SensorValue0.3		;
iTank1Sensor1ValueTemp.5		:= 			IusiTank1SensorValue0.2		;
iTank1Sensor1ValueTemp.6		:= 			IusiTank1SensorValue0.1		;
iTank1Sensor1ValueTemp.7		:= 			IusiTank1SensorValue0.0		;                                					
iTank1Sensor1ValueTemp.8		:= 			IusiTank1SensorValue1.7		;
iTank1Sensor1ValueTemp.9		:= 			IusiTank1SensorValue1.6		;
iTank1Sensor1ValueTemp.10		:= 			IusiTank1SensorValue1.5		;
iTank1Sensor1ValueTemp.11		:= 			IusiTank1SensorValue1.4		;
iTank1Sensor1ValueTemp.12		:= 			IusiTank1SensorValue1.3		;
iTank1Sensor1ValueTemp.13		:= 			IusiTank1SensorValue1.2		;
													
iTank1Sensor1Value.0			:=			iTank1Sensor1ValueTemp.13	;
iTank1Sensor1Value.1			:=			iTank1Sensor1ValueTemp.12	;													
iTank1Sensor1Value.2			:=			iTank1Sensor1ValueTemp.11	;													
iTank1Sensor1Value.3			:=			iTank1Sensor1ValueTemp.10	;													
iTank1Sensor1Value.4			:=			iTank1Sensor1ValueTemp.9	;													
iTank1Sensor1Value.5			:=			iTank1Sensor1ValueTemp.8	;													
iTank1Sensor1Value.6			:=			iTank1Sensor1ValueTemp.7	;													
iTank1Sensor1Value.7			:=			iTank1Sensor1ValueTemp.6	;													
iTank1Sensor1Value.8			:=			iTank1Sensor1ValueTemp.5	;													
iTank1Sensor1Value.9			:=			iTank1Sensor1ValueTemp.4	;													
iTank1Sensor1Value.10			:=			iTank1Sensor1ValueTemp.3	;													
iTank1Sensor1Value.11			:=			iTank1Sensor1ValueTemp.2	;													
iTank1Sensor1Value.12			:=			iTank1Sensor1ValueTemp.1	;													
iTank1Sensor1Value.13			:=			iTank1Sensor1ValueTemp.0	;													

(***Skalownaie wartości zadanej na 1-100%************)
(*Filtrowanie sygnału jeżeli włączony jest CIP*)
IF bCIP THEN
	fbFilterExiTank1Sensor1Value(
				rIn:=				INT_TO_REAL(iTank1Sensor1Value), 
				tTimeConstant:= 	T#50MS, 
				rOut=>				);
	VIS.iTank1LevelSensorValue := REAL_TO_INT(fbFilterExiTank1Sensor1Value.rOut);	
ELSE
//	VIS.iTank1LevelSensorValue := iTank1Sensor1Value;
END_IF
(****Koniec skalownaie wartości zadanej na 1-100%****)
																																												
bTank1SensorDiagnosis										:= NOT P00_PneumaticValves.fbiTank1LevelSensorValue.bError;

IF uTank1LevelSetpoint>290 THEN
	uTank1LevelSetpoint:=290;//Zabezpieczenie przed zbyt wielka nastawą
END_IF

//ZAŁĄCZANIE POMPY OD ZADANEJ WARTOŚCI
IF VIS.lrDispencer1DoseVolumeShow > 450 THEN
	tonTank1LevelLowConductiveSensor( IN:=VIS.iTank1LevelSensorValue < UINT_TO_INT(uTank1LevelSetpoint) AND bTank1SensorDiagnosis AND NOT bExEnable, PT:=T#1S);
ELSE
	tonTank1LevelLowConductiveSensor( IN:=VIS.iTank1LevelSensorValue < UINT_TO_INT(uTank1LevelSetpoint) AND bTank1SensorDiagnosis AND NOT bExEnable, PT:=T#10S);	
END_IF


IF tonTank1LevelLowConductiveSensor.Q THEN
	bTank1LevelLowConductiveSensor := TRUE;
ELSE
	bTank1LevelLowConductiveSensor := FALSE;
END_IF
(****************************KONIEC ZBIORNIK 1***********************************************************)

(*Przypisane na stałe*)

//VIS.uTank2LevelSetpointShow:=75; // bylo 120
IF VIS.uTank2LevelSetpointShow > 201 THEN
	VIS.uTank2LevelSetpointShow := 100;
END_IF

(**************************** ZBIORNIK 2***********************************************************)
                     
	iTank2Sensor1ValueTemp.0		:= 			IusiTank2SensorValue0.7		;
	iTank2Sensor1ValueTemp.1		:= 			IusiTank2SensorValue0.6		;
	iTank2Sensor1ValueTemp.2		:= 			IusiTank2SensorValue0.5		;
	iTank2Sensor1ValueTemp.3		:= 			IusiTank2SensorValue0.4		;
	iTank2Sensor1ValueTemp.4		:= 			IusiTank2SensorValue0.3		;
	iTank2Sensor1ValueTemp.5		:= 			IusiTank2SensorValue0.2		;
	iTank2Sensor1ValueTemp.6		:= 			IusiTank2SensorValue0.1		;
	iTank2Sensor1ValueTemp.7		:= 			IusiTank2SensorValue0.0		;                                					
	iTank2Sensor1ValueTemp.8		:= 			IusiTank2SensorValue1.7		;
	iTank2Sensor1ValueTemp.9		:= 			IusiTank2SensorValue1.6		;
	iTank2Sensor1ValueTemp.10		:= 			IusiTank2SensorValue1.5		;
	iTank2Sensor1ValueTemp.11		:= 			IusiTank2SensorValue1.4		;
	iTank2Sensor1ValueTemp.12		:= 			IusiTank2SensorValue1.3		;
	iTank2Sensor1ValueTemp.13		:= 			IusiTank2SensorValue1.2		;
														
	iTank2Sensor1Value.0			:=			iTank2Sensor1ValueTemp.13	;
	iTank2Sensor1Value.1			:=			iTank2Sensor1ValueTemp.12	;													
	iTank2Sensor1Value.2			:=			iTank2Sensor1ValueTemp.11	;													
	iTank2Sensor1Value.3			:=			iTank2Sensor1ValueTemp.10	;													
	iTank2Sensor1Value.4			:=			iTank2Sensor1ValueTemp.9	;													
	iTank2Sensor1Value.5			:=			iTank2Sensor1ValueTemp.8	;													
	iTank2Sensor1Value.6			:=			iTank2Sensor1ValueTemp.7	;													
	iTank2Sensor1Value.7			:=			iTank2Sensor1ValueTemp.6	;													
	iTank2Sensor1Value.8			:=			iTank2Sensor1ValueTemp.5	;													
	iTank2Sensor1Value.9			:=			iTank2Sensor1ValueTemp.4	;													
	iTank2Sensor1Value.10			:=			iTank2Sensor1ValueTemp.3	;													
	iTank2Sensor1Value.11			:=			iTank2Sensor1ValueTemp.2	;													
	iTank2Sensor1Value.12			:=			iTank2Sensor1ValueTemp.1	;													
	iTank2Sensor1Value.13			:=			iTank2Sensor1ValueTemp.0	;													
	     
	(****Koniec skalownaie wartości zadanej na 1-100%****)
																																													
	bTank2SensorDiagnosis										:= NOT P00_PneumaticValves.fbiTank2LevelSensorValue.bError;

VIS.iTank2LevelSensorValue := iTank2Sensor1Value;	
	//ZAŁĄCZANIE POMPY OD ZADANEJ WARTOŚCI
//ZAŁĄCZANIE POMPY OD ZADANEJ WARTOŚCI
tonTank2LevelLowConductiveSensor( IN:=VIS.iTank2LevelSensorValue < UINT_TO_INT(uTank2LevelSetpoint) AND bTank2SensorDiagnosis AND NOT bExEnable, PT:=T#10S);
IF tonTank2LevelLowConductiveSensor.Q THEN
	bTank2LevelLowConductiveSensor := TRUE;
ELSE
	bTank2LevelLowConductiveSensor := FALSE;
END_IF
(****************************KONIEC ZBIORNIK 2***********************************************************)
END_ACTION

END_PROGRAM

(* stored: Version 1.1.0.1, ProductVersion 3.1.4026.13, FileIdentifier d50d6037687b46f22e098546b82334a100513d86, FileSignature 503c8ac5e249d78a99b3994921ef9ca129f32bf2e5ff1e8a21448ab4fe391d8272f2ffde9ab533e29120458550d6bc2873ea0507c68f64024da1e0fbfca64326cd5b36d4aee5a3c6e833697d831217e7eb658b69d34f15e4659cd756f2764bc4b949c127a13f274f38d1863d5b7dc75c80e742b2da7f3433b790de6e76fadffa358de700520ab56d8c8c5b6b7c62e8ff286e273c0b710e880e01e527c620cd71716d44eb4e9e1fc28c2362cd4a5484849210036eab0f07e9e9c1bea449ea7da39715066e2837b48eb7c609d05fe3177bd865d4310566c162c9cda064ad069817ca35766b2b475783cb3751a79a735f772e84c61309fb247bcf8de6327f6a7d0a
   POU P02_Dispencers: Id {d18c9b08-0ea9-4290-b431-6012e40a7c42}, SpecialFunc None
   Folder Dispencers: Id {aadee575-c276-4c3c-bcc7-6cf7cbb6c968}
   Folder DragStation: Id {4d802563-ab1b-46f6-befc-83e0f58e6083}
   Action aAntyColision: Id {315e4bb4-aa5f-4e48-ab15-87139dc9aa85}
   Action aCleaning: Id {f43e1c2b-3ef0-4d3a-8c7f-5b838c16b51e}
   Action aDispencer1: Id {0727b44a-8ec0-48d7-9d8c-66266bdaf399}
   Action aDispencer2: Id {db692009-14e8-4e4e-b600-655f4ca62978}
   Action aDispencer3: Id {4659f61e-5469-4cdc-a47e-a272f9e38873}
   Action aDispencer4: Id {0870676a-f880-4dec-9c92-dd294b270645}
   Action aDispencerCatch1: Id {ed201ba5-ed0a-46ef-8f7e-97bd882110c8}
   Action aDispencerCatch2: Id {022bba26-aaf8-491b-a9fb-b5a79e1de30c}
   Action aDispencerCatch3: Id {27aa668a-23db-41ca-845f-4a14ab45c708}
   Action aDispencerCatch4: Id {79ddfb87-01f4-4821-a2b7-bda2094050d9}
   Action aDispencerCatchPressure: Id {632ee484-6d47-43c9-8e69-0d090586637f}
   Action aDispencerDragStation: Id {33c160db-6ae3-4b54-b3bb-6501bf9d7ab8}
   Action aDispencersCatchWarnings: Id {d045c6c7-7674-4a07-969f-500b189c7131}
   Action aDispencersDragStationLeadActuators: Id {79802fc1-c9f3-4f66-b9b4-dedada596750}
   Action aDispencersEnable: Id {829fd3c9-a08a-443d-96b7-070ce115508d}
   Action aDispencersLiftersAfter: Id {a58fae64-7f41-476f-a4ab-2c3806ccc5cd}
   Action aDispencersLiftersBefore: Id {b7e2a927-5d6b-48d2-8b94-faaa255de5e6}
   Action aDispencersManualMode: Id {99741657-8c1f-4213-837d-0f73592a900a}
   Action aDosingChartHMI: Id {6ed426e7-d3d6-4849-858a-05d12632c302}
   Action aDropCatcher: Id {991e144f-fa88-4315-83df-06a1aea5e4af}
   Action aExSensor: Id {b050d5d6-743a-42ba-a681-a20e3ab65ebf}
   Action aLevelSensorCalibration: Id {d743aade-5b8f-44d1-ad83-11fd653f6f76}
   Action aLimits: Id {0c9ded22-8f11-454f-b7a2-17d9156a4a50}
   Action aTankHeating: Id {42bc75ac-e89c-4286-a329-413e6ac24517}
   Action aTanks: Id {7144bf1b-2159-4de2-b2fa-88db0a1a1b53}
   Action aTanksRainbowMode: Id {d2886ec9-8203-4999-8224-a84053232340}
   Action aTankWarning: Id {9bd88b64-dbf1-4daf-abb5-8fc3d3bbfab6}
   Action aTDRMassSensor: Id {8b699bd6-9e4d-4f2e-ac0b-11e5c1a46999} *)
